PROGRAM PRG_ComputeMovingSetPoint
VAR
END_VAR

END_PROGRAM

(* stored: Version 1.1.0.1, ProductVersion 3.1.4022.7
   POU PRG_ComputeMovingSetPoint: Id {83a101db-fed2-42da-9701-7b259ab0243c}, SpecialFunc None *)
